// TwinCAT 3 PLC project RoomController
// ProgramVersion: 3.1.4023.0
// libraries:
//   Tc2_Standard, * (Beckhoff Automation GmbH)
//   Tc2_System, * (Beckhoff Automation GmbH)
//   Tc3_Module, * (Beckhoff Automation GmbH)
// project tree:
//   DUTs/ stAi4CH.TcDUT (not stored), stRoomData.TcDUT (not stored)
//   GVLs/ IO.TcGVL
//   / PlcTask.TcTTO
//   POUs/ fbIntValueSimulation.TcPOU (not stored), Hardware_Simulation.TcPOU (not stored), MAIN.TcPOU (not stored)
// real-time tasks:
//   TASK PlcTask: cycle T#10ms, priority 20, ADS port 350
// I/O:
//   DEVICE Device 1 (EtherCAT) (disabled), AmsNetId 172.20.10.2.2.1
//     Term 1 (EK1200) [EK1200-5000 EtherCAT Power supply (2A E-Bus)]
//       Term 2 (EL3164) [EL3164 4Ch. Ana. Input 0-10V]
//       Term 3 (EL9011) [EL9011 End Terminal]
// variable links:
//   RoomController/RoomController Instance <-> Device 1 (EtherCAT)/Term 1 (EK1200)/Term 2 (EL3164)
//     PlcTask Inputs/IO.hwAirDataIN.CH{1..4} <-> AI Standard Channel {1..4}/Value  (4 links)

CONFIGURATION RoomController
    RESOURCE PLC ON TwinCAT3
        TASK PlcTask(INTERVAL := T#10ms, PRIORITY := 20);
        PROGRAM MAIN WITH PlcTask : MAIN;
    END_RESOURCE
END_CONFIGURATION

// ---- GVLs/IO.TcGVL
{attribute 'qualified_only'}
VAR_GLOBAL
	hwAirDataIN : stAi4CH;
END_VAR
